{attribute addProperty BoxType "AT2000-0233-0022"}
{attribute addProperty Id "CC_Inputs_14_ChAT %I*CC_Inputs_14_Ch_5FB71CBE240300CC_Outputs_14_ChAT %Q*CC_Outputs_14_Ch_8D55E481240300WcStateAT %I*WcState_98A4DF7520.250InfoDataAT %I*InfoData_0BDED7BF144180"}
{attribute addProperty CRC "2331747689"}
{attribute addProperty SizeInBites "626"}
{attribute addProperty SizeInBytes "78.25"}
TYPE AT2000_15405010 :
STRUCT
	{attribute addProperty Name "CC_Inputs_14_Ch"}
	CC_Inputs_14_Ch : CC_Inputs_14_Ch_5FB71CBE;
	{attribute addProperty Name "CC_Outputs_14_Ch"}
	CC_Outputs_14_Ch : CC_Outputs_14_Ch_8D55E481;
	{attribute addProperty Name "WcState"}
	WcState : WcState_98A4DF75;
	{attribute addProperty Name "InfoData"}
	InfoData : InfoData_0BDED7BF;
END_STRUCT
END_TYPE

(* stored: Version 1.2.0.0, ProductVersion 3.1.4024.9
   DUT AT2000_15405010: Id {0e112fb0-4bb0-4c02-950c-bd78466776ee} *)
